TYPE ST_TaskData :
STRUCT
	CycleTime 		: LREAL;
	LastExecTime	: LREAL;
	SystemLatency	: LREAL; 
END_STRUCT
END_TYPE

(* stored: Version 1.1.0.1
   DUT ST_TaskData: Id {70495082-e389-491c-99f6-aa0630dd23e0} *)
